// Alarm information structure, containing all the informations requoired
TYPE ST_AlarmInfo :
STRUCT
	Name			: Tc2_System.T_MaxString;	// Name of the alarm
	Id				: T_ArrayIndexer;			// Id of the alarm
	Message			: Tc2_System.T_MaxString;	// Message of the alarm
	IsActive		: BOOL;						// Active state (TRUE = currently active, FALSE = not active)
	IsAcknowledged	: BOOL;						// Acknowledge state of the alarm
	Level			: E_AlarmLevel;				// Alarm level
	TimeInfos		: ST_AlarmTimeInfos;		// Time informations (activated, acknowldiged, deactivated)
END_STRUCT
END_TYPE

(* stored: Version 1.1.0.1
   DUT ST_AlarmInfo: Id {463a7f24-175c-0f47-0a80-135f9f8b1f98} *)
